Universal Robots PolyScope program: home.urp

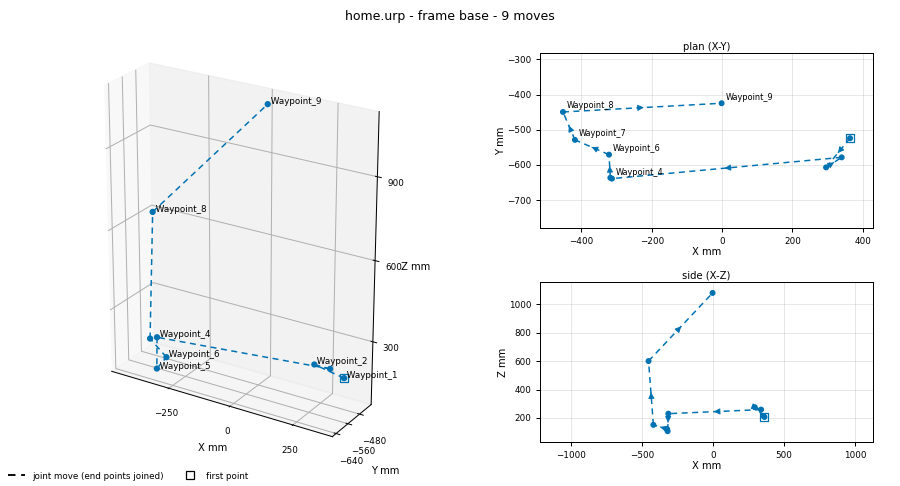
[picture p0: tool path of home.urp in frame base, 9 of 9 moves have a stored position in this frame; points joined in program order, loops and branches not executed]
Program home (installation=default directory=/programs/yutongxie createdIn=5.12.6.1102099 lastSavedIn=5.12.6.1102099 robotSerialNumber=20215500597)
Calibrated DH parameters: a=[0.000193, -0.066673, -0.391568, -0.000012, 0.00005, 0]; d=[0.162643, -472.05677, 465.132521, 7.058239, 0.099746, 0.099582]; alpha=[1.571116, 0.00089, 0.003862, 1.569269, -1.569248, 0]; deltaTheta=[0, -1.413394, 7.628392, 0.068187, 0, -0.000001]
Robot Program (runOnlyOnce=true)
  MoveJ speed 60 deg/s, acceleration 80 deg/s^2 (useActiveTCP=true) feature=Base
    Waypoint Waypoint_1: TCP in base x=363.663 y=-524.199 z=206.962 mm, rx=-2.1294 ry=-0.3551 rz=-1.9842 rad; joints [85.735, -55.086, 83.182, -38.364, -22.833, 98.803] deg; TCP offset x=0 y=0 z=191.5 mm, rx=0 ry=0 rz=0 rad
    Waypoint Waypoint_2: TCP in base x=295.566 y=-607.114 z=275.807 mm, rx=1.9177 ry=-0.5577 rz=1.835 rad; joints [79.622, -77.376, 106.632, -24.67, 23.846, 84.189] deg
    Waypoint Waypoint_3: TCP in base x=339.935 y=-578.68 z=258.958 mm, rx=1.3941 ry=0.8461 rz=0.793 rad; joints [83.724, -76.894, 110.447, -33.514, 23.368, -2.071] deg
    Waypoint Waypoint_4: TCP in base x=-313.373 y=-639.151 z=230.336 mm, rx=1.5684 ry=0.0065 rz=-0.0199 rad; joints [31.573, -71.696, 108.788, -37.63, 32.159, -0.47] deg
    Waypoint Waypoint_5: TCP in base x=-317.933 y=-636.765 z=106.824 mm, rx=1.6062 ry=0.0362 rz=-0.0573 rad; joints [31.143, -59.467, 112.115, -49.047, 32.154, -6.437] deg
    URCap Gripper (Robotiq_Grippers, Robotiq Inc.) dataModel(position=0.0, force=0.0, speed=0.0, positionInDouble=0.0, forceInDouble=0.0, speedInDouble=0.0, slaveIds=[9], blocking=true)
    Waypoint Waypoint_6: TCP in base x=-321.652 y=-570.974 z=121.67 mm, rx=1.5454 ry=-0.0127 rz=-0.0059 rad; joints [22.931, -64.134, 121.712, -61.447, 23.811, 3.804] deg
    Waypoint Waypoint_7: TCP in base x=-418.552 y=-528.934 z=151.411 mm, rx=1.5718 ry=0.1294 rz=0.1857 rad; joints [12.622, -56.77, 99.435, -40.976, 1.237, 0.39] deg
    Waypoint Waypoint_8: TCP in base x=-452.592 y=-449.623 z=600.853 mm, rx=1.1637 ry=1.2667 rz=-1.1886 rad; joints [3.038, -92.19, 90.115, -89.816, -0.567, 0.027] deg
    Waypoint Waypoint_9: TCP in base x=-1.546 y=-424.817 z=1080.554 mm, rx=-0.0044 ry=-2.2185 rz=2.2204 rad; joints [0.001, -90, -0.001, -90, -0.002, -0.001] deg
    URCap Gripper (Robotiq_Grippers, Robotiq Inc.) dataModel(position=100.0, force=0.0, speed=0.0, positionInDouble=100.0, forceInDouble=0.0, speedInDouble=0.0, slaveIds=[9], blocking=true)
